Staubli VAL3: onF5Event.pgx

program onF5Event(bool& x_bSave[] (dimensions=1))
begin
  // look if the bButton is enable
  if bButton[4]
    //
    // Wizard
    call setPallet(x_bSave)
    // rebuild the list
    call buildList()
  endIf
end
